Fanuc KAREL source: kt00260.KL

-- PROVISIONAL review KL for V770-1; original PC SHA256 225f52f37e16d7542625a37d8850a7c227ee8b25434f6f2ccb7396d7a3f68fa3
-- Incomplete behavior may be omitted. Consult companion uncertainty JSON. Do not deploy.
PROGRAM KT00260
%NOLOCKGROUP
VAR
  I1 : INTEGER
  OUT : BOOLEAN
-- UNRESOLVED_DECL H2 type=002017
BEGIN
  -- UNRESOLVED_PC offsets 5-16; opcodes 2E,23
  -- UNRESOLVED_PC offsets 21-35; opcodes 2E,22,9D,33,B4
  -- UNRESOLVED_PC offsets 40-62; opcodes 21,22,9D,33,B3,57,23
  -- UNRESOLVED_PC offsets 67-71; opcodes 7F
END KT00260
